// TIA Portal V20 export
FUNCTION_BLOCK "FB_Maintenance"   // FB471, SCL
{ S7_Optimized_Access := 'TRUE' }
// stored: AutoNumber false, MemoryReserve 100, SetENOAutomatically false
   VAR_INPUT
      iIncrementEnable { ExternalAccessible := 'False'; ExternalVisible := 'False'; ExternalWritable := 'False'} : Bool;
      iID { ExternalAccessible := 'False'; ExternalVisible := 'False'; ExternalWritable := 'False'} : Int;
   END_VAR
   VAR_IN_OUT
      ioOPC : "UDT_OPC_Maintenance";
      ioAlarm { ExternalAccessible := 'False'; ExternalVisible := 'False'; ExternalWritable := 'False'} : Bool;   // Alarme (100% atteint)
      ioWarning { ExternalAccessible := 'False'; ExternalVisible := 'False'; ExternalWritable := 'False'} : Bool;   // Avertissement (80% atteint)
   END_VAR
   VAR
      sElement { ExternalAccessible := 'False'; ExternalVisible := 'False'; ExternalWritable := 'False'} : "UDT_MaintenanceElement";
   END_VAR
   VAR_TEMP
      tUsagePercent : Real;
      tAdjustedIncrement : Bool;
   END_VAR
BEGIN
   REGION Description header 
       //==================================================================================
       // POSALUX Swiss SA / (C) Copyright 2024
       //----------------------------------------------------------------------------------
       // Title: Gestion_Temps_Fonctionnement
       // Comment/Function: Cette fonction  assure le suivi du temps de fonctionnement
       //                   des équipements et génère des alertes basées sur
       //                   leur utilisation. Elle incrémente le temps de fonctionnement
       //                   selon l'unité définie (minute, heure, jour), calcule le
       //                   pourcentage d'utilisation par rapport à un seuil d'alarme, et
       //                   gère les avertissements et alarmes en fonction de ce pourcentage
       //
       // Author: Gowsigan SRITHARAN
       // Engineering: TIA Portal v17
       //----------------------------------------------------------------------------------
       // Change log table:
       // Version  | Date     | Expert in charge | Changes applied
       // ---------|----------|------------------|------------------------------------
       // 00.00.01 | 20241120 | GSR              | First released version
       // ---------|----------|------------------|------------------------------------
       // 01.01.01 | 20241219 | FMI              | Utilisation d'un flanc montant du clock1Hz pour compter en secondes
       // ==================================================================================
   END_REGION

   REGION Incrementation du temps en secondes
       IF "DB_Impulsion".sRT_Clock_1Hz.Q AND #iIncrementEnable THEN
           #sElement.RunTimeSec := #sElement.RunTimeSec + 1;
       END_IF;
   END_REGION

   REGION Incrementation du temps en fonction du type unité
       CASE #sElement.TimeUnit OF
           0:
               #sElement.RunTime := #sElement.RunTimeSec / 60.0;     // Affichage runtime en minutes
           1:
               #sElement.RunTime := #sElement.RunTimeSec / 3600.0;   // Affichage runtime en heures
           2:
               #sElement.RunTime := #sElement.RunTimeSec / 86400.0;  // Affichage runtime en jours
       END_CASE;

   END_REGION

   REGION Gestion des warnings et alarmes    
       // Définir l'état de l'alarme et des avertissements en fonction du pourcentage d'utilisation
       #ioAlarm   := #sElement.RunTime >= #sElement.AlarmThreshold;                      // Alarme si utilisation atteint ou dépasse le seuil d'alarme
       #ioWarning := #sElement.RunTime >= #sElement.WarningThreshold AND NOT #ioAlarm;   // Avertissement si utilisation dépasse le seuil d'avertissement sans alarme active
   END_REGION

   REGION OPC Communication
       #ioOPC.Elapsed := #sElement.RunTime;
       #ioOPC.WarningThreshold := #sElement.WarningThreshold;
       #ioOPC.Period := #sElement.AlarmThreshold;
       #ioOPC.Id := #iID;
       #sElement.ResetRunTime :=#ioOPC.Reset;
       #ioOPC.Reset := FALSE;
   END_REGION

   REGION Reset du compteur
       IF #sElement.ResetRunTime THEN
           #sElement.RunTimeSec := 0;       // Reset du compteur de temps de fonctionnement
           #sElement.ResetRunTime := FALSE;
       END_IF;
   END_REGION
END_FUNCTION_BLOCK
